FUNCTION_BLOCK HandshakeRequester (* Handshake pattern demo: Plug / Requester role *)
  (* Standard: 61499-2; Description: Copyright (c) 2026 Meisterschulen am Ostbahnhof This program and the accompanying materials are made available under the terms of the Eclipse Public License 2.0 which is available at https://www.eclipse.org/legal/epl-2.0/ SPDX-License-Identifier: EPL-2.0 *)
  (* Version 1.3, 2026-08-31, Franz Höpfinger, Meisterschulen am Ostbahnhof, Fixed INIT handling: dedicated Init/Initialized/DeInit states with INIT[TRUE=QI]/INIT[FALSE=QI] guards (per TemplateBasic.fbt), instead of resetting counters on every re-entry to idle *)
  (* Version 1.2, 2026-08-31, Franz Höpfinger, Meisterschulen am Ostbahnhof, EVENT_HS EventInputs/EventOutputs swapped so the Requester is now a Plug (more natural layout) - back to Plugs here *)
  (* Version 1.1, 2026-08-31, Franz Höpfinger, Meisterschulen am Ostbahnhof, Handshake design pattern (IEC 61499 primer course, Module 6, Valeriy Vyatkin), demo Requester *)
  (* Version 1.0, 2026-08-31, Franz Höpfinger, Meisterschulen am Ostbahnhof, initial version, wrongly declared as Plug - fixed to Socket *)
  PACKAGE Meins::DesingPatterns::HandshakePattern;
  (* Documentation:
  Requester ("client") side of the Handshake design pattern (IEC 61499 primer course, Module 6, Valeriy Vyatkin, slide 72).
   Uses the dataless adapter::events::Handshake::EVENT_HS adapter as a Plug: on START it sends a REQ and reports DONE once the matching CNF comes back; whenever an unsolicited IND arrives it answers with RSP and reports NOTIFIED.
   Per the adapter's own declaration, the Plug side is the one that fires REQ/RSP and reacts to CNF/IND - i.e. the Plug plays the client/Requester role here, the Socket plays the server/Responder role. See HandshakePattern.md in this folder for the full write-up.
  *)
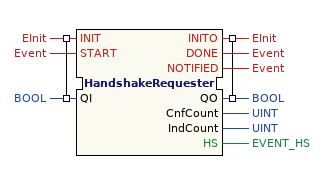
  EVENT_INPUT
    INIT : EInit WITH QI; (* Initialization Request *)
    START; (* Demo: fire a REQ towards the Responder *)
  END_EVENT
  EVENT_OUTPUT
    INITO : EInit WITH QO; (* Initialization Confirm *)
    DONE; (* A CNF was received for the last REQ *)
    NOTIFIED; (* An IND was received and answered with RSP *)
  END_EVENT
  VAR_INPUT
    QI : BOOL; (* Input event qualifier *)
  END_VAR
  VAR_OUTPUT
    QO : BOOL; (* Output event qualifier *)
    CnfCount : UINT; (* Number of CNF received (demo counter) *)
    IndCount : UINT; (* Number of IND received / RSP sent (demo counter) *)
  END_VAR
  PLUGS
    HS : adapter::types::bidirectional::Handshake::EVENT_HS; (* Handshake plug: sends REQ/RSP, receives CNF/IND *)
  END_PLUGS
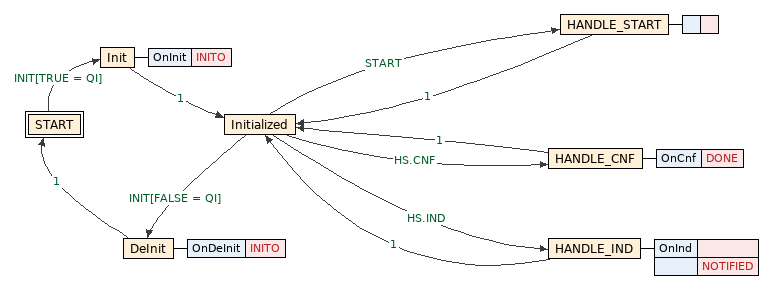
  EC_STATES
    START; (* Uninitialized *)
    Init : OnInit -> INITO; (* Initialization *)
    Initialized; (* Idle, ready to react *)
    DeInit : OnDeInit -> INITO; (* De-initialization *)
    HANDLE_START; (* Send a REQ *)
    HANDLE_CNF : OnCnf -> DONE; (* A CNF arrived, report DONE *)
    HANDLE_IND : OnInd, -> NOTIFIED; (* An IND arrived, answer with RSP and report NOTIFIED *)
  END_STATES
  EC_TRANSITIONS
    START TO Init := INIT[TRUE = QI];
    Init TO Initialized := 1;
    Initialized TO DeInit := INIT[FALSE = QI];
    DeInit TO START := 1;
    Initialized TO HANDLE_START := START;
    HANDLE_START TO Initialized := 1;
    Initialized TO HANDLE_CNF := HS.CNF;
    HANDLE_CNF TO Initialized := 1;
    Initialized TO HANDLE_IND := HS.IND;
    HANDLE_IND TO Initialized := 1;
  END_TRANSITIONS
  ALGORITHM OnInit IN ST: (* Reset demo counters *)
CnfCount := 0;
IndCount := 0;
QO := QI;
  END_ALGORITHM
  ALGORITHM OnDeInit IN ST: (* De-initialize *)
QO := FALSE;
  END_ALGORITHM
  ALGORITHM OnCnf IN ST: (* Count a received CNF *)
CnfCount := CnfCount + 1;
  END_ALGORITHM
  ALGORITHM OnInd IN ST: (* Count a received IND, about to answer with RSP *)
IndCount := IndCount + 1;
  END_ALGORITHM
END_FUNCTION_BLOCK
